(* CoDeSys 2.3 export: F_WRITE_WB_VALVELS_CFG.EXP *)

(* POU FUN/PARAMETERS/F_WRITE_WB_VALVELS_CFG, ST *)
FUNCTION F_WRITE_WB_VALVELS_CFG : BOOL
VAR_INPUT
	sHead : STRING;
	wSize   :DWORD;
	pBuffer :POINTER TO BYTE;
END_VAR
VAR_IN_OUT
	wPos     : DWORD;
	stConfig : ST_WB_VALVE_LS_CFG;
END_VAR
VAR
END_VAR
F_ADD_STRINGX3_TO_BUFFER( S1:= '$n#', S2:= sHead, S3:=' - Parameters:$n', wSize := wSize, pBuffer := pBuffer, wPos := wPos );

F_ADD_STRINGX4_TO_BUFFER( S1:= CONCAT(sHead, '_TimeMax'   ), S2:='$t', S3:= REAL_TO_STRING( stConfig.TimeMax  ), S4:='$n', wSize := wSize, pBuffer := pBuffer, wPos := wPos );
F_ADD_STRINGX4_TO_BUFFER( S1:= CONCAT(sHead, '_PushTime'  ), S2:='$t', S3:= REAL_TO_STRING( stConfig.PushTime ), S4:='$n', wSize := wSize, pBuffer := pBuffer, wPos := wPos );
F_ADD_STRINGX4_TO_BUFFER( S1:= CONCAT(sHead, '_PushPress' ), S2:='$t', S3:= REAL_TO_STRING( stConfig.PushP    ), S4:='$n', wSize := wSize, pBuffer := pBuffer, wPos := wPos );

F_ADD_STRINGX4_TO_BUFFER( S1:= CONCAT(sHead, '_TgtLS_Half' ), S2:='$t', S3:= REAL_TO_STRING( stConfig.TgtLS_Half ), S4:='$n', wSize := wSize, pBuffer := pBuffer, wPos := wPos );
F_ADD_STRINGX4_TO_BUFFER( S1:= CONCAT(sHead, '_LS_DB'      ), S2:='$t', S3:= REAL_TO_STRING( stConfig.LS_DB      ), S4:='$n', wSize := wSize, pBuffer := pBuffer, wPos := wPos );

F_ADD_STRINGX4_TO_BUFFER( S1:= CONCAT(sHead, '_HP'        ), S2:='$t', S3:= BYTE_TO_STRING( stConfig.HP       ), S4:='$n', wSize := wSize, pBuffer := pBuffer, wPos := wPos );
END_FUNCTION
